FUNCTION_BLOCK AX_BOOL_TO_X (* Composite FB for convert BOOL to AX *)
  (* Standard: 61499-2 *)
  (* Version 1.0, 2024-04-24, franz *)
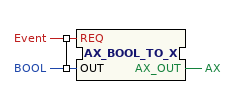
  EVENT_INPUT
    REQ WITH OUT; (* Initialization Request *)
  END_EVENT
  VAR_INPUT
    OUT : BOOL;
  END_VAR
  PLUGS
    AX_OUT : AX;
  END_PLUGS
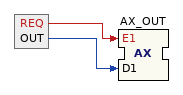
  EVENT_CONNECTIONS
    REQ TO AX_OUT.E1;
  END_CONNECTIONS
  DATA_CONNECTIONS
    OUT TO AX_OUT.D1;
  END_CONNECTIONS
END_FUNCTION_BLOCK
